(* IEC 61131-3 sources: programs/VI-54/VI-54_20171205/VI-54_20171205/Stations/PLC_VI54/VI-54_171014/Class/Recipe_Machine, 1 file *)

(* ---- Recipe_Machine.st ---- *)
(*!
<Class
	Name               = "Recipe_Machine"
	Revision           = "0.0"
	RealtimeTask       = "false"
	CyclicTask         = "false"
	BackgroundTask     = "false"
	Sigmatek           = "false"
	OSInterface        = "false"
	HighPriority       = "false"
	Automatic          = "false"
	UpdateMode         = "Prescan"
	SharedCommandTable = "true"
	Objectsize         = "(810,420)">
	<Channels>
		<Server Name="LineSpeed" Visualized="true" Initialize="false" WriteProtected="false" Retentive="false"/>
		<Server Name="Max_AccDec" Visualized="true" Initialize="false" WriteProtected="true" Retentive="false"/>
		<Server Name="Max_Speed" Visualized="true" Initialize="false" WriteProtected="true" Retentive="false"/>
		<Client Name="MotionValues" Required="true" Internal="false"/>
	</Channels>
	<Separators>
		<Servers>
			<SepChn Position="2"/>
		</Servers>
	</Separators>
	<Network Name="Recipe_Machine">
		<!-- List of Components in this network -->
		<Components>
			<Object
				Name       = "_base"
				Class      = "RecipeBase"
				Position   = "(218,120)"
				Visualized = "false">
				<Channels>
					<Server Name="Comm"/>
					<Client Name="MainRecipe"/>
				</Channels>
			</Object>
		</Components>
		<Comments>
		</Comments>
		<!-- List of Connections in this network -->
		<Connections>
			<Connection Source="this.Comm" Destination="_base.Comm" Vertices="(690,210),(518,210),"/>
			<Connection Source="_base.MainRecipe" Destination="this.MainRecipe" Vertices="(218,210),(38,210),"/>
		</Connections>
		<!-- Headerfiles -->
		<Options>
		</Options>
	</Network>
</Class>
*)
#pragma using RecipeBase

Recipe_Machine : CLASS
: RecipeBase
  //Servers:
	Max_Speed 	: SvrCh_DINT;
	Max_AccDec 	: SvrCh_DINT;
	LineSpeed 	: SvrCh_DINT;
  //Clients:
	MotionValues 	: CltChCmd__LMC_MotorInfo;
  //Variables:
  //Functions:

	FUNCTION VIRTUAL GLOBAL Init;

	FUNCTION VIRTUAL GLOBAL LineSpeed::Write
		VAR_INPUT
			input (EAX) 	: DINT;
		END_VAR
		VAR_OUTPUT
			result (EAX) 	: DINT;
		END_VAR;
  //Tables:
	FUNCTION @STD
		VAR_OUTPUT
			ret_code	: CONFSTATES;
		END_VAR;
	FUNCTION GLOBAL TAB @CT_;
END_CLASS;

#pragma usingLtd _LMC_MotorInfo

FUNCTION VIRTUAL GLOBAL Recipe_Machine::Init

  // open init methode of baseclass
  RecipeBase::Init();

  Max_Speed   := to_dint(to_real MotionValues.MaxSpeed ToMperMin);
  Max_AccDec  := to_dint(to_real MotionValues.MaxAccDec ToMperSec2);

END_FUNCTION

FUNCTION VIRTUAL GLOBAL Recipe_Machine::LineSpeed::Write
	VAR_INPUT
		input (EAX) 	: DINT;
	END_VAR
	VAR_OUTPUT
		result (EAX) 	: DINT;
	END_VAR

	LineSpeed := input;
  ReceptPtr^.Machine.LineSpeed := LineSpeed;
	result := LineSpeed;

END_FUNCTION
